# EPICS substitutions: evrSupport/Db/ioc/evrPatternTO20.substitutions
#
# Pattern records
file evrPatternAll.db {
#	    Device        ,  SLC Pattern Check LNK    , EVR/Trigger
#	                                                  Links
  pattern { DEVICE        ,        LINK4              , LINK5 , LINK6 , TREF }
	{ IOC:TO20:IM01 ,"IOC:TO20:IM01:FANOUTSLC"      ,  ""   ,"IOC:TO20:IM01:FANOUT", 1.03E06 }
}
file evrEventAll.db {
  pattern { DEVICE        }
	  { IOC:TO20:IM01 }
}
